// Mitsubishi GX Developer project: 240707_trafficLight   PLC: FX series

PROGRAM MAIN
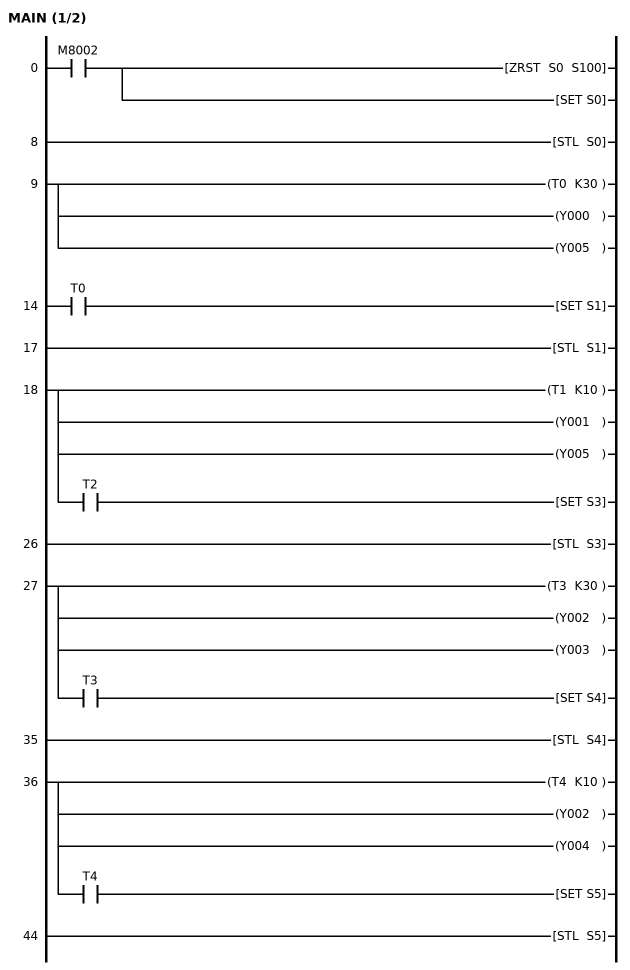
0     LD      M8002
      ZRST    S0 S100
      SET     S0
8     STL     S0
9     OUT     T0 K30
      OUT     Y000
      OUT     Y005
14    LD      T0
      SET     S1
17    STL     S1
18    OUT     T1 K10
      OUT     Y001
      OUT     Y005
      AND     T2
      SET     S3
26    STL     S3
27    OUT     T3 K30
      OUT     Y002
      OUT     Y003
      AND     T3
      SET     S4
35    STL     S4
36    OUT     T4 K10
      OUT     Y002
      OUT     Y004
      AND     T4
      SET     S5
44    STL     S5
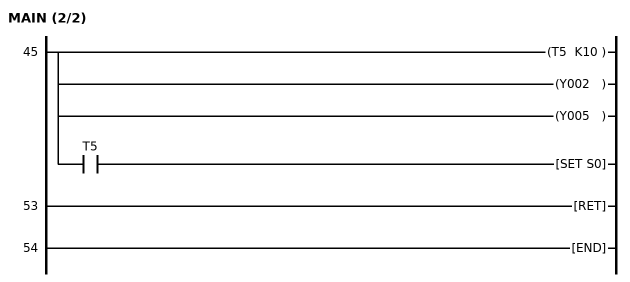
45    OUT     T5 K10
      OUT     Y002
      OUT     Y005
      AND     T5
      SET     S0
53    RET
54    END
END_PROGRAM
